{attribute 'qualified_only'}

TYPE stackerLoadDisplayStates :
(
	dStStartingUp 			:= 1000,
	dStStandBy,
	dStStackerIsReseting,
	dStAxisNotConfigured,
	dStRemotePalletManually,
	dStFixerCylinderDidNotOpen,
	dStFixerCylinderDidNotClose,
	dStLock1CylinderDidNotOpen,
	dStLock1CylinderDidNotClose,
	dStLock2CylinderDidNotOpen,
	dStLock2CylinderDidNotClose,
	dStFestoDriveError,
	dStAxisInitMoveTakesTooLong,
	dStWaitForPalletsLoading, 
	dStLoadPallets, 
	dStPalletLoadMoveTakesTooLong,
	dStWaitForPallet,
	dStPalletMoveTakesTooLong,
	dStReleaseEmptyPallet,
    dStThereIsNoPalletOnTop,
	dStStationIsStopped,
	dStWaitForNextStep

	
)DINT;
END_TYPE

(* stored: Version 1.1.0.1, ProductVersion 3.1.4024.3
   DUT stackerLoadDisplayStates: Id {94844f0d-83aa-41a4-be1f-5ba67d9a6932} *)
